Staubli VAL3: PositionUpdate.pgx

program PositionUpdate()
begin
  while true
    jCurrentJoint=herej()
    jCurrentJointError=getPositionErr()
    pCurrentPosition=jointToPoint(flange,world,jCurrentJoint-jCurrentJointError)
    //pCurrentPosition = here(flange, world)
    delay(0.01)
  endWhile
end
